PROGRAM MAIN
VAR
END_VAR

END_PROGRAM

(* stored: Version 1.1.0.1
   POU MAIN: Id {e11ac494-e854-4cf7-8266-0956a115f8c6} *)
